// TIA Portal V20 export
VAR_GLOBAL   // PLC tag table "Global"
END_VAR
VAR_GLOBAL CONSTANT   // user constants
   UNIT01 : Int := 0;   // Unit 1
   NO_OF_UNITS : Int := 1;   // Highest value of unit (Counting starts from 0)
   NO_OF_PANELS : Int := 1;   // Highest value of HMI(Counting starts from 1)
   NO_OF_EM : UDInt := 16;   // Highest value of EMs
END_VAR
